FUNCTION_BLOCK FB83
TITLE = 'process_F3'
AUTHOR : CB

VAR
	tmp : BOOL;
END_VAR


BEGIN


NETWORK
TITLE =
//
//	process/process_F3/KNEAD1PROC
CALL FC82 (combE := 1);
CALL FB82,	DB82;
CALL FC82 (combE := 0);




END_FUNCTION_BLOCK
